TYPE STATE:
    STRUCT
        curTime: REAL;
        dvar_M_a: DINT;
    END_STRUCT;
END_TYPE
